RESOURCE_TYPE DE2_115
  (* Standard: 61499-2 *)
  (* Version 0.1, 2016-00-31, hpea485, UOA *)
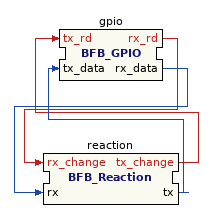
  FBS
    gpio : BFB_GPIO;
    reaction : BFB_Reaction;
  END_FBS
  EVENT_CONNECTIONS
    gpio.rx_rd TO reaction.rx_change;
    reaction.tx_change TO gpio.tx_rd;
  END_CONNECTIONS
  DATA_CONNECTIONS
    gpio.rx_data TO reaction.rx;
    reaction.tx TO gpio.tx_data;
  END_CONNECTIONS
END_RESOURCE_TYPE
